RoboDK station: multi pass welding with change in height.rdk

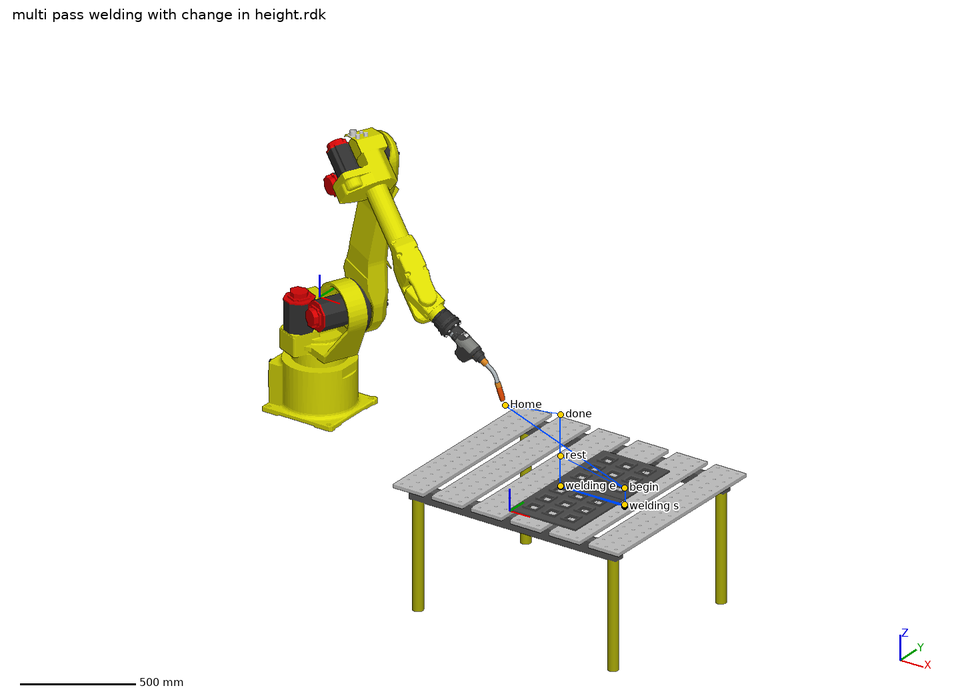
[picture v0: the station drawn from its stored meshes, robots at their saved joint values, targets as dots, program paths as lines]
Station multi pass welding with change in height (saved by RoboDK 5.9.2). Poses are relative to the parent item; angles as X-Y-Z fixed-axis rotations.
  - frame Fanuc ARC Mate 120iB Base at (-540, 0, 505) mm
    - robot Fanuc ARC Mate 120iB: 6 axes
        modified DH rows (alpha deg, a mm, theta deg, d mm): 0, 0, 0, 525; -90, 150, -90, 0; 0, 770, 0, 0; -90, 100, 0, 740; 90, 0, 0, 0; -90, 0, 0, 100
        base shift (0, 0, -525) mm
        joint limits [-170, -80, -170, -200, -140, -450] to [170, 170, 250, 200, 140, 450]; home [0, 0, 0, 0, 0, 0]; saved at [-23.563, 8.476, -41.451, -106.099, -20.017, 301.011]
      - tool Fronius MTB500i Welding Gun, TCP at (86, 0, 461.5) mm, rotated rx 0 ry 36 rz 0 deg, size 139 x 105 x 455.9 mm
  - object Table 1200x1000mm (Welding) at (780, 0, 0) mm, size 1193.8 x 965.2 x 609.6 mm, geometry from Table-1200x1000mm-Welding.sld
  - frame Frame 2 at (750, -410, 0) mm
    - object plate 1 at (0, 0, 0) mm, size 350 x 350 x 20 mm, geometry from Pallete .step
    - object plate 2 at (0, 360, 0) mm, size 350 x 350 x 20 mm, geometry from Pallete .step
    - target Home (Cartesian target) at (-58.15, 52.89, 470.6) mm, rotated rx -179.42 ry 20.57 rz -179.8 deg; joints [-30.481, -5.248, -41.931, -99.83, -25.158, 299.21] of Fanuc ARC Mate 120iB
    - target begin (Cartesian target) at (359.45, 357.84, 68.27) mm, rotated rx -179.42 ry 20.57 rz -179.8 deg; joints [-2.265, 49.247, -56.086, -175.87, -22.699, 357.887] of Fanuc ARC Mate 120iB
    - target welding s (Cartesian target) at (359.45, 357.84, -21.73) mm, rotated rx -179.42 ry 20.57 rz -179.8 deg; joints [-2.265, 54.419, -60.355, -176.485, -26.959, 358.565] of Fanuc ARC Mate 120iB
    - target welding e (Cartesian target) at (19.46, 357.84, -21.73) mm, rotated rx -179.42 ry 20.57 rz -179.8 deg; joints [-3.13, 42.465, -80.587, -176.843, -47.174, 360.029] of Fanuc ARC Mate 120iB
    - target rest (Cartesian target) at (19.46, 357.84, 128.27) mm, rotated rx -179.42 ry 20.57 rz -179.8 deg; joints [-3.13, 30.409, -69.764, -176.095, -36.371, 359.03] of Fanuc ARC Mate 120iB
    - target s 1 (Cartesian target) at (359.45, 357.84, -21) mm, rotated rx -179.42 ry 20.57 rz -179.8 deg; joints [-2.265, 54.376, -60.323, -176.481, -26.926, 358.561] of Fanuc ARC Mate 120iB
    - target s 2 (Cartesian target) at (359.45, 357.84, -20) mm, rotated rx -179.42 ry 20.57 rz -179.8 deg; joints [-2.265, 54.317, -60.278, -176.476, -26.882, 358.555] of Fanuc ARC Mate 120iB
    - target s 3 (Cartesian target) at (359.45, 357.84, -19) mm, rotated rx -179.42 ry 20.57 rz -179.8 deg; joints [-2.265, 54.258, -60.233, -176.47, -26.837, 358.549] of Fanuc ARC Mate 120iB
    - target s 4 (Cartesian target) at (359.45, 357.84, -18) mm, rotated rx -179.42 ry 20.57 rz -179.8 deg; joints [-2.265, 54.199, -60.188, -176.465, -26.792, 358.542] of Fanuc ARC Mate 120iB
    - target s 5 (Cartesian target) at (359.46, 357.84, -17) mm, rotated rx -179.42 ry 20.57 rz -179.8 deg; joints [-2.265, 54.14, -60.143, -176.46, -26.747, 358.536] of Fanuc ARC Mate 120iB
    - target s 6 (Cartesian target) at (359.46, 357.84, -15) mm, rotated rx -179.42 ry 20.57 rz -179.8 deg; joints [-2.265, 54.022, -60.053, -176.448, -26.657, 358.524] of Fanuc ARC Mate 120iB
    - target s 7 (Cartesian target) at (359.45, 357.84, -13) mm, rotated rx -179.42 ry 20.57 rz -179.8 deg; joints [-2.265, 53.904, -59.963, -176.437, -26.567, 358.511] of Fanuc ARC Mate 120iB
    - target e 1 (Cartesian target) at (19.45, 357.84, -21) mm, rotated rx -179.42 ry 20.57 rz -179.8 deg; joints [-3.13, 42.404, -80.539, -176.841, -47.126, 360.025] of Fanuc ARC Mate 120iB
    - target e 2 (Cartesian target) at (19.45, 357.84, -20) mm, rotated rx -179.42 ry 20.57 rz -179.8 deg; joints [-3.13, 42.322, -80.473, -176.837, -47.06, 360.02] of Fanuc ARC Mate 120iB
    - target e 3 (Cartesian target) at (19.46, 357.84, -19) mm, rotated rx -179.42 ry 20.57 rz -179.8 deg; joints [-3.13, 42.24, -80.407, -176.834, -46.995, 360.015] of Fanuc ARC Mate 120iB
    - target e 4 (Cartesian target) at (19.46, 357.84, -19) mm, rotated rx -179.42 ry 20.57 rz -179.8 deg; joints [-3.13, 42.24, -80.407, -176.834, -46.995, 360.015] of Fanuc ARC Mate 120iB
    - target e 5 (Cartesian target) at (19.45, 357.84, -18) mm, rotated rx -179.42 ry 20.57 rz -179.8 deg; joints [-3.13, 42.157, -80.341, -176.831, -46.929, 360.01] of Fanuc ARC Mate 120iB
    - target e 6 (Cartesian target) at (19.45, 357.84, -17) mm, rotated rx -179.42 ry 20.57 rz -179.8 deg; joints [-3.13, 42.075, -80.275, -176.827, -46.863, 360.005] of Fanuc ARC Mate 120iB
    - target e 7 (Cartesian target) at (19.45, 357.84, -17) mm, rotated rx -179.42 ry 20.57 rz -179.8 deg; joints [-3.13, 42.075, -80.275, -176.827, -46.863, 360.005] of Fanuc ARC Mate 120iB
    - target done (Cartesian target) at (19.46, 357.84, 327) mm, rotated rx -179.42 ry 20.57 rz -179.8 deg; joints [-3.13, 16.508, -53.48, -173.267, -20.151, 355.852] of Fanuc ARC Mate 120iB
  - program Prog1 (51 instructions, listed below)
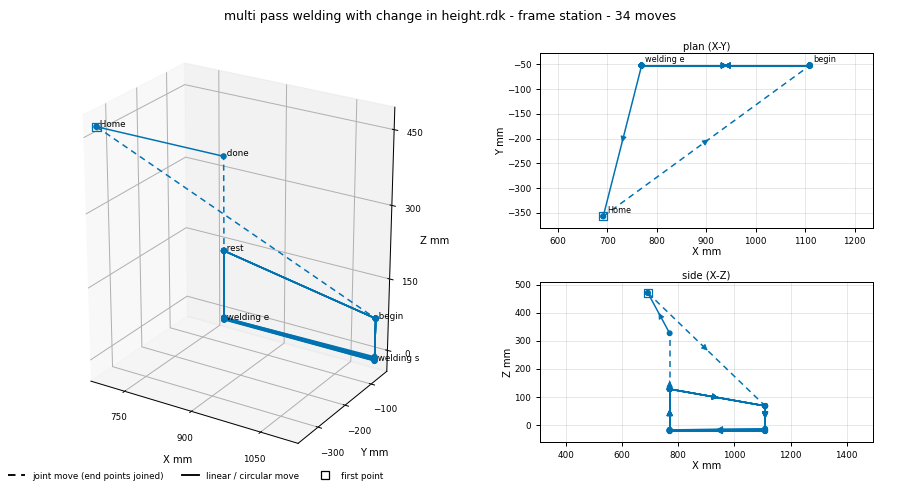
[picture p0: tool path of multi pass welding with change in height.rdk in frame station, 34 of 34 moves have a stored position in this frame; points joined in program order, loops and branches not executed]

--- program Prog1 (robot Fanuc ARC Mate 120iB) ---
  Set Ref.: Frame 2
  Set Tool: Fronius MTB500i Welding Gun
  MoveJ (Home)
  MoveJ (begin)
  MoveL (welding s)
  Pause 500 ms
  MoveL (welding e)
  Pause 500 ms
  MoveL (rest)
  MoveL (begin)
  Pause 500 ms
  MoveL (s 1)
  MoveL (e 1)
  MoveL (rest)
  Pause 500 ms
  MoveL (begin)
  Pause 500 ms
  MoveL (s 2)
  MoveL (e 2)
  MoveL (rest)
  Pause 500 ms
  MoveL (begin)
  Pause 500 ms
  MoveL (s 3)
  MoveL (e 3)
  MoveL (rest)
  Pause 500 ms
  MoveL (begin)
  Pause 500 ms
  MoveL (s 4)
  MoveL (e 4)
  MoveL (rest)
  Pause 500 ms
  MoveL (begin)
  Pause 500 ms
  MoveL (s 5)
  MoveL (e 5)
  MoveL (rest)
  Pause 500 ms
  MoveL (begin)
  Pause 500 ms
  MoveL (s 6)
  MoveL (e 6)
  MoveL (rest)
  Pause 500 ms
  MoveL (begin)
  Pause 500 ms
  MoveL (s 7)
  MoveL (e 7)
  MoveJ (done)
  MoveL (Home)
